{attribute 'hide'}
FUNCTION F_HwSetAddrInfo_29bit : ST_CanData_29bit
VAR_INPUT
	stInput: ST_CanHeader;
END_VAR

F_HwSetAddrInfo_29bit.nCobid := 16#3FFFFFFF AND stInput.nCobid;

IF (stInput.nCobid > 16#7FF AND NOT stInput.bExtendedAddress) THEN // check cobid and extended address flags is set correctly
	stInput.bExtendedAddress := TRUE;//fix issue
END_IF

F_HwSetAddrInfo_29bit.nCobid.31 := stInput.bExtendedAddress;//sets extended address flag, if set raw can message will have 29bit for identification on the wire.

F_HwSetAddrInfo_29bit.nCobid.30 := stInput.bRTR;// sets RTR bit

IF (stInput.nMsgLength > 8) THEN
	F_HwSetAddrInfo_29bit.nLength := 8;
ELSE
	F_HwSetAddrInfo_29bit.nLength := stInput.nMsgLength;
END_IF

END_FUNCTION

(* stored: Version 1.1.0.1, ProductVersion 3.1.4024.12
   POU F_HwSetAddrInfo_29bit: Id {88cecfba-8168-0632-201d-e7b81bcd29c5}, SpecialFunc None *)
